# B&R Automation Studio project Lab1
Automation Studio 4.5.2.102

## Configuration Config1

CPU 4PP065.0571-P74, AutomationRuntime D4.52, Build 4.1.2, Vc V4.52.0, Safety 1.6

### Hardware
```
4PP065_0571_P74 : 4PP065.0571-P74 v1.1.2.0
  Connector IF5:
    ActivateDevice = 1
  ConfigurationID = lab1v1_Config1
  Simulation = 1
```

## Logical view

Binary libraries used (declarations not repeated): operator, runtime, astime, AsIecCon

### Library Logical/Libraries/Library (ANSIC)

#### Library.fun
```iecst
{REDUND_ERROR} {REDUND_UNREPLICABLE} FUNCTION_BLOCK FB_Motor (*TODO: Add your comment here*) (*$GROUP=User,$CAT=User,$GROUPICON=User.png,$CATICON=User.png*)
	VAR_INPUT
		u : {REDUND_UNREPLICABLE} REAL;
	END_VAR
	VAR_OUTPUT
		w : {REDUND_UNREPLICABLE} REAL;
		phi : {REDUND_UNREPLICABLE} REAL;
	END_VAR
	VAR
		integrator : {REDUND_UNREPLICABLE} FB_Integrator;
		Tm : {REDUND_UNREPLICABLE} REAL;
		ke : {REDUND_UNREPLICABLE} REAL;
		dt : {REDUND_UNREPLICABLE} REAL;
	END_VAR
END_FUNCTION_BLOCK

{REDUND_ERROR} FUNCTION_BLOCK FB_Integrator (*TODO: Add your comment here*) (*$GROUP=User,$CAT=User,$GROUPICON=User.png,$CATICON=User.png*)
	VAR_INPUT
		in : {REDUND_UNREPLICABLE} REAL;
	END_VAR
	VAR
		out : {REDUND_UNREPLICABLE} REAL;
		dt : {REDUND_UNREPLICABLE} REAL;
		prev_value : REAL;
	END_VAR
END_FUNCTION_BLOCK

{REDUND_ERROR} FUNCTION_BLOCK FB_Regulator (*TODO: Add your comment here*) (*$GROUP=User,$CAT=User,$GROUPICON=User.png,$CATICON=User.png*)
	VAR_INPUT
		e : {REDUND_UNREPLICABLE} REAL;
	END_VAR
	VAR_OUTPUT
		u : REAL;
	END_VAR
	VAR
		integrator : FB_Integrator;
		k_p : REAL;
		k_i : REAL;
		iyOld : REAL;
		dt : REAL;
		max_abs_value : REAL;
	END_VAR
END_FUNCTION_BLOCK
```

#### FB_Motor.c
```c
#include <bur/plctypes.h>
#ifdef __cplusplus
  extern "C"
  {
#endif
#include "Library.h"
#ifdef __cplusplus
  };
#endif

void FB_Motor(struct FB_Motor* inst)
{
	REAL a = inst->u / inst->ke - inst->w;
	REAL b = a / inst->Tm;

	inst->integrator.in = b;
	FB_Integrator(&inst->integrator);

	inst->w = inst->integrator.out;
}
```

#### FB_Regulator.c
```c
#include <bur/plctypes.h>
#ifdef __cplusplus
  extern "C"
  {
#endif
#include "Library.h"
#ifdef __cplusplus
  };
#endif

void FB_Regulator(struct FB_Regulator* inst)
{
	//vremennye peremennye
	REAL a = inst->e * inst ->k_p;
	REAL b = inst->e * inst ->k_i;
  	//ogranichenie napryazeniya

	a = a > inst->max_abs_value ? inst ->max_abs_value : a;
	a = a < -inst ->max_abs_value ? -inst ->max_abs_value : a;

	inst->integrator.in = b + inst->iyOld;

	FB_Integrator(&inst->integrator);

	REAL sum = a + inst->integrator.out;
	inst->u = sum;

	//ogranichenie napryazeniya
	inst->u = inst->u > inst->max_abs_value ? inst->max_abs_value : inst->u;
	inst->u = inst->u < -inst->max_abs_value ? inst->max_abs_value : inst->u;

	inst->iyOld = inst->u - sum;
}
```

### Program Logical/Program (ANSIC)

#### Main.c - Cyclic code
```c
#include <bur/plctypes.h>

#ifdef _DEFAULT_INCLUDES
#include <AsDefault.h>
#endif

void _INIT ProgramInit(void)
{
	fb_motor1.dt = 0.01;
	fb_motor1.ke = 0.24;
	fb_motor1.Tm = 0.1;
	fb_motor1.u = 0;
	fb_motor1.integrator.dt=0.01;

	fb_motor2.dt = 0.01;
	fb_motor2.ke = 0.24;
	fb_motor2.Tm = 0.1;
	fb_motor2.u = 0;
	fb_motor2.integrator.dt=0.01;

	fb_controller.dt = 0.01;
	fb_controller.integrator.dt = 0.01;
	fb_controller.k_i = 0.2;
	fb_controller.k_p = 0.78;
	fb_controller.max_abs_value = 24.0;

	Speed = 0;
	counter = 0;
	Enable = 1;
}

void _CYCLIC ProgramCyclic(void)
{
	if (Enable)
	{
		if(counter == 200)
		{
			Speed = 0;
			counter = 0;
		}
		else if (counter == 50)
		{
			Speed = 50;
		}
		counter++;

		fb_controller.e = Speed - fb_motor1.w;
		FB_Regulator(&fb_controller);

		fb_motor1.u = fb_controller.u;
		FB_Motor(&fb_motor1);

		fb_motor2.u = Speed * fb_motor2.ke;
		FB_Motor(&fb_motor2);
	}
}

void _EXIT ProgramExit(void)
{

}
```

#### Variables.var - Local variables
```iecst
VAR
	Enable : BOOL;
	counter : INT;
	fb_motor1 : FB_Motor;
	fb_controller : FB_Regulator;
	fb_motor2 : FB_Motor;
	Speed : REAL;
END_VAR
```

Listed in the project but not available here: Logical/Program/Types.typ
